KUKA KRL program: eki_communication.src, eki_communication.dat

--- eki_communication.src ---
&ACCESS RVO
&REL 4
&PARAM DISKPATH = KRC:\R1\Program\ROS
DEF eki_communication ( )
   ; Software License Agreement (BSD License)
   ;
   ; Copyright (c) 2022, Kuka Robotics Corp
   ; All rights reserved.
   ;
   ; Redistribution and use in source and binary forms, with or without
   ; modification, are permitted provided that the following conditions are met:
   ;
   ;      * Redistributions of source code must retain the above copyright
   ;        notice, this list of conditions and the following disclaimer.
   ;      * Redistributions in binary form must reproduce the above copyright
   ;        notice, this list of conditions and the following disclaimer in the
   ;        documentation and/or other materials provided with the distribution.
   ;      * Neither the name of the copyright holder, nor the names of its
   ;        contributors may be used to endorse or promote products derived
   ;        from this software without specific prior written permission.
   ;
   ; THIS SOFTWARE IS PROVIDED BY THE COPYRIGHT HOLDERS AND CONTRIBUTORS "AS IS"
   ; AND ANY EXPRESS OR IMPLIED WARRANTIES, INCLUDING, BUT NOT LIMITED TO, THE
   ; IMPLIED WARRANTIES OF MERCHANTABILITY AND FITNESS FOR A PARTICULAR PURPOSE
   ; ARE DISCLAIMED. IN NO EVENT SHALL THE COPYRIGHT OWNER OR CONTRIBUTORS BE
   ; LIABLE FOR ANY DIRECT, INDIRECT, INCIDENTAL, SPECIAL, EXEMPLARY, OR
   ; CONSEQUENTIAL DAMAGES (INCLUDING, BUT NOT LIMITED TO, PROCUREMENT OF
   ; SUBSTITUTE GOODS OR SERVICES; LOSS OF USE, DATA, OR PROFITS; OR BUSINESS
   ; INTERRUPTION) HOWEVER CAUSED AND ON ANY THEORY OF LIABILITY, WHETHER IN
   ; CONTRACT, STRICT LIABILITY, OR TORT (INCLUDING NEGLIGENCE OR OTHERWISE)
   ; ARISING IN ANY WAY OUT OF THE USE OF THIS SOFTWARE, EVEN IF ADVISED OF THE
   ; POSSIBILITY OF SUCH DAMAGE.

END

GLOBAL DEF EKI_ServerInit()

   InterfaceName[] = "EkiKSSinterface"

END

GLOBAL DEF EKI_ServerStart()
   decl eki_status eki_ret

   ; Init connection flag - will be set TRUE internally by EKI after connection is made
   $flag[ROS_EKI_Conn_Flag] = FALSE
   ; Init data recv flag - will be set TRUE internally by EKI after data is received
   $flag[ROS_EKI_Recv_Flag] = FALSE

   ; TODO: check ret values
   eki_ret = EKI_Init(InterfaceName[])
   eki_ret = EKI_Open(InterfaceName[])
END

DEF EKI_ServerReset()
   decl eki_status eki_ret
   eki_ret = EKI_Clear(InterfaceName[])
   EKI_ServerStart()
END

; Tries to read received elements from buffer.
GLOBAL DEF EKI_ReceiveData(cmd: OUT)
   DECL EKI_Status eki_ret
   DECL EKI_Status eki_ret_req
   DECL Command cmd

   ; Init cmd
   cmd.cmd_str[] = "None"
   cmd.cmdID = -1
   cmd.control_mode = -1

   ; Verify a valid connection
   IF (NOT Connected()) THEN
      WAIT SEC 0.012
      RETURN
   ENDIF

   ; Skip processing if no data received.
   IF (NOT $FLAG[ROS_EKI_Recv_Flag]) THEN
      WAIT SEC 0.012
      RETURN
   ENDIF

   ; Reset flag immediately after msg notification
   $FLAG[ROS_EKI_Recv_Flag] = FALSE

   eki_ret_req = eki_checkbuffer(InterfaceName[], "External/@REQTYPE")

   IF eki_ret_req.buff > 0 THEN

      eki_ret_req = eki_getString(InterfaceName[], "External/@REQTYPE", cmd.cmd_str[])
      eki_ret = eki_getINT(InterfaceName[], "External/@ID", cmd.cmdID)
      eki_ret = eki_getINT(InterfaceName[], "External/@ControlMode", cmd.control_mode)

      ; Nothing valid in buffer
   ELSE
      MsgNotify("No valid data received")
      WAIT SEC 0.012
   ENDIF

END

GLOBAL DEF HandleConnection()
   IF (Connected() <> connection_flag) THEN
      connection_flag = Connected()
      IF (Connected() == TRUE) THEN
         MsgNotify("External client connected")
      ELSE
         MsgNotify("External client disconnected")
         EKI_ServerReset()
      ENDIF
   ENDIF
END

GLOBAL DEF PublishEvent()
   DECL EKI_STATUS eki_ret
   DECL INT event_int
   DECL CHAR event_msg[64]

   IF GetEvent() <> #None THEN
      IF Connected() == FALSE THEN
         MsgNotify("External client is not connected when trying to send event")
         RETURN
      ENDIF

      ; TODO make this nicer if possible
      SWITCH last_event
         CASE #Started
            event_int = 0
         CASE #Stopped
            event_int = 1
         CASE #Cancelled
            event_int = 2
         CASE #ResetOK
            event_int = 3
         CASE #Error
            event_int = 4
         CASE #Connected
            event_int = 5
         CASE #SwitchOK
            event_int = 6
            SWITCH GetControlMode()
               CASE #JointPosition
                  event_msg[] = "joint position control"
               CASE #CartPosition
                  event_msg[] = "cartesian position control"
               DEFAULT
                  event_msg[] = "inactive control"
            ENDSWITCH
            eki_ret = eki_setString(InterfaceName[], "Robot/Event/@Message", event_msg[])
         CASE #Invalid
            event_int = 7
         DEFAULT
            event_int = 8
      ENDSWITCH

      eki_ret = eki_setInt(InterfaceName[], "Robot/Event/@EventID", event_int)
      eki_ret = eki_setInt(InterfaceName[], "Robot/Status/@Mode", 1) ; TODO: op mode

      ; Transmit the current Run Mode
      eki_ret = eki_setInt(InterfaceName[], "Robot/Status/@ControlMode", 1) ; TODO

      ; Send the message
      ;eki_ret = eki_send(InterfaceName[], "Robot/Status")
      eki_ret = eki_send(InterfaceName[], "Robot/Event")

      ; Reset event
      SetEvent(#None)
   ENDIF
END

GLOBAL DEFFCT BOOL Connected()
   RETURN $FLAG[ROS_EKI_Conn_Flag]
ENDFCT

GLOBAL DEF SetEvent(event: IN)
   DECL EventType event
   last_event = event
END

GLOBAL DEFFCT EventType GetEvent()
   RETURN last_event
ENDFCT

--- eki_communication.dat ---
&ACCESS RV
&REL 4
&PARAM DISKPATH = KRC:\R1\Program\ROS
DEFDAT eki_communication
    STRUC EventTypeTuple EventType event_type, INT event_type_int

    CONST CHAR INTERFACE_NAME[64]
    INTERFACE_NAME[] = "EkiKSSinterface"
    CONST CHAR INTERFACE_VERSION[16]
    INTERFACE_VERSION[] = "1.0.0"
    CONST INT ROS_EKI_CONN_FLAG = 105
    CONST INT ROS_EKI_RECV_FLAG = 110

    ; FOLD Helper constant for decoding axis type information
    CONST CHAR AXIS_TYPE_MAP[5, 16]
    AXIS_TYPE_MAP[1,] = "LINEAR"
    AXIS_TYPE_MAP[2,] = "NOT_USED" ; Not used
    AXIS_TYPE_MAP[3,] = "ROTATIONAL"
    AXIS_TYPE_MAP[4,] = "NOT_USED" ; Not used
    AXIS_TYPE_MAP[5,] = "ENDLESS"
    ; ENDFOLD

    ; FOLD Constants for easier mapping of event types to integers
    DECL CONST EventTypeTuple EVENT_TYPE_TUPLES[12]
    EVENT_TYPE_TUPLES[1] = { event_type #STARTED, event_type_int 0 }
    EVENT_TYPE_TUPLES[2] = { event_type #STOPPED, event_type_int 1 }
    EVENT_TYPE_TUPLES[3] = { event_type #CANCELLED, event_type_int 2 }
    EVENT_TYPE_TUPLES[4] = { event_type #RESET_OK, event_type_int 3 }
    EVENT_TYPE_TUPLES[5] = { event_type #ERROR, event_type_int 4 }
    EVENT_TYPE_TUPLES[6] = { event_type #CONNECTED, event_type_int 5 }
    EVENT_TYPE_TUPLES[7] = { event_type #SWITCH_OK, event_type_int 6 }
    EVENT_TYPE_TUPLES[8] = { event_type #INVALID, event_type_int 7 }
    EVENT_TYPE_TUPLES[9] = { event_type #NONE, event_type_int 8 }
    EVENT_TYPE_TUPLES[10] = { event_type #DRIVES_TURNED_ON, event_type_int 9 }
    EVENT_TYPE_TUPLES[11] = { event_type #DRIVES_TURNED_OFF, event_type_int 10 }
    EVENT_TYPE_TUPLES[12] = { event_type #CYCLE_TIME_CHANGED, event_type_int 11 }
    ; ENDFOLD

    DECL BOOL connection_flag = FALSE
    DECL EventType last_event = #NONE
ENDDAT
